// SIMATIC S7-200 project (STEP 7-Micro/WIN), CPU 221 REL 01.10

SYMBOL_TABLE IO
I顶升气缸下位          I0.0
I顶升气缸上位          I0.1
I上工位检测           I0.2
I本工位检测           I0.3
I下工位检测           I0.4
I毛刷2             I0.5
I扳手监控2           I0.6
I自动手动旋钮          I0.7
I放行按钮1           I1.0
I复位按钮            I1.1
I放行按钮2           I1.2
I急停按钮            I1.3
I_12             I1.4
I_13             I1.5
I取料监控6           I2.0
I取料监控5           I2.1
I取料监控4           I2.2
I取料监控3           I2.3
I取料监控2           I2.4
I取料监控1           I2.5
I形状辅具2           I2.6
I定长辅具2           I2.7
I_24             I3.0
I定长辅具1           I3.1
I形状辅具1           I3.2
I_27             I3.3
I毛刷1             I3.4
I扳手监控1           I3.5
I_30             I3.6
I_31             I3.7
Q下阻挡器放行          Q0.0
Q顶升气缸下降          Q0.1
Q上阻挡器放行          Q0.2
Q顶升气缸上升          Q0.3
Q_2              Q0.4
Q_3              Q0.5
Q_4              Q0.6
Q_5              Q0.7
Q_6              Q1.0
Q_7              Q1.1
Q_8              Q1.2
Q_9              Q1.3
Q_10             Q1.4
Q_11             Q1.5
Q_12             Q1.6
Q_13             Q1.7
Q_14             Q2.0
Q_15             Q2.1
Q_16             Q2.2
Q_17             Q2.3
Q_18             Q2.4
Q_19             Q2.5
Q_20             Q2.6
Q_21             Q2.7
Q红灯              Q3.0
Q黄灯              Q3.1
Q绿灯              Q3.2
Q蜂鸣器             Q3.3
Q_26             Q3.4
Q_27             Q3.5
Q_28             Q3.6
Q_29             Q3.7
END_SYMBOL_TABLE

SYMBOL_TABLE M
M上阻挡器放行          M100.0
M下阻挡器放行          M100.1
M顶升气缸上升          M100.2
M顶升气缸下降          M100.3
M104             M100.4
M105             M100.5
M106             M100.6
M107             M100.7
M通讯正常            M1000.0
M联线状态            M1000.2
工位RFID读取触发       M2000.0
工位RFID读取完成       M2000.1
工位上序合格           M2000.2
工位上序不合格          M2000.3
工位本序已做           M2000.4
工位放行中            M2001.0
本序合格             M2001.1
本序不合格            M2001.2
M自动工步            MD3000
END_SYMBOL_TABLE
